TYPE STMTargetVelocity :
STRUCT
	velocity : INT;
	acceleration : UINT;
	deceleration : UINT;
END_STRUCT
END_TYPE

(* stored: Version 1.1.0.1, ProductVersion 3.1.4024.11
   DUT STMTargetVelocity: Id {7d15a199-c2c3-4eb7-9448-0c9a45ce7a50} *)
